{attribute addProperty BoxType "IODEVICETYPE_ETHERCATPROT"}
{attribute addProperty Id "Beckhoff_ER1xxxBeckhoff_ER1xxx_F144525A3562445.25Beckhoff_ER2xxxBeckhoff_ER2xxx_C2CD7B256706838.25Beckhoff_ER3xxxBeckhoff_ER3xxx_0B6E7FA92872359Beckhoff_ER4xxxBeckhoff_ER4xxx_C7805EB066282.75Beckhoff_ER5xxxBeckhoff_ER5xxx_1B1665E350262.75Beckhoff_ER6xxxBeckhoff_ER6xxx_39EF444F3498437.25Beckhoff_ER7xxxBeckhoff_ER7xxx_A258BD7D2934366.75Beckhoff_ER8xxxBeckhoff_ER8xxx_BCCF515741051.25SyncUnitsSyncUnits_CAB22D3B19524.375InputsInputs_C75D3FEC1280160OutputsOutputs_47D1E803848106InfoDataInfoData_E9F65A829612"}
{attribute addProperty CRC "3544190561"}
{attribute addProperty SizeInBites "23565"}
{attribute addProperty SizeInBytes "2945.625"}
TYPE EtherCAT_Master_ERxxxx_D3400E61 :
STRUCT
	{attribute addProperty Name "Beckhoff_ER1xxx"}
	Beckhoff_ER1xxx : Beckhoff_ER1xxx_F144525A;
	{attribute addProperty Name "Beckhoff_ER2xxx"}
	Beckhoff_ER2xxx : Beckhoff_ER2xxx_C2CD7B25;
	{attribute addProperty Name "Beckhoff_ER3xxx"}
	Beckhoff_ER3xxx : Beckhoff_ER3xxx_0B6E7FA9;
	{attribute addProperty Name "Beckhoff_ER4xxx"}
	Beckhoff_ER4xxx : Beckhoff_ER4xxx_C7805EB0;
	{attribute addProperty Name "Beckhoff_ER5xxx"}
	Beckhoff_ER5xxx : Beckhoff_ER5xxx_1B1665E3;
	{attribute addProperty Name "Beckhoff_ER6xxx"}
	Beckhoff_ER6xxx : Beckhoff_ER6xxx_39EF444F;
	{attribute addProperty Name "Beckhoff_ER7xxx"}
	Beckhoff_ER7xxx : Beckhoff_ER7xxx_A258BD7D;
	{attribute addProperty Name "Beckhoff_ER8xxx"}
	Beckhoff_ER8xxx : Beckhoff_ER8xxx_BCCF5157;
	{attribute addProperty Name "SyncUnits"}
	SyncUnits : SyncUnits_CAB22D3B;
	{attribute addProperty Name "Inputs"}
	Inputs : Inputs_C75D3FEC;
	{attribute addProperty Name "Outputs"}
	Outputs : Outputs_47D1E803;
	{attribute addProperty Name "InfoData"}
	InfoData : InfoData_E9F65A82;
END_STRUCT
END_TYPE

(* stored: Version 1.2.0.0, ProductVersion 3.1.4024.9
   DUT EtherCAT_Master_ERxxxx_D3400E61: Id {1885ac0f-3299-4bae-a679-e872c07c4bcb} *)
